// TIA Portal project "LIMIT" (V16)

(* hardware
DEVICE "S7-1200 station_1"  S7-1200 Station
   slot 0: "Rack_0"  S7-1200 Rack  Rack  V1.0
   slot 1: "PLC_1"  CPU 1212C AC/DC/Rly  6ES7 212-1BE40-0XB0  V4.4
*)

// ===== PLC "PLC_1"  CPU 1212C AC/DC/Rly =====

VAR_GLOBAL   // PLC tag table "Default tag table"
   "START" AT %I0.0 : Bool;
   "STOP" AT %I0.1 : Bool;
   "M1" AT %Q0.0 : Bool;
   "X" AT %M0.0 : Bool;
   "TM" AT %M0.1 : Bool;
   "L1" AT %I0.2 : Bool;
   "L2" AT %I0.3 : Bool;
   "L3" AT %I0.4 : Bool;
   "OFF" AT %M1.1 : Bool;
   "M2" AT %Q0.1 : Bool;
   "Tag_1" AT %M2.0 : Bool;
END_VAR

// folder: System blocks/Program resources

DATA_BLOCK "T"   // DB1
{ S7_Optimized_Access := 'TRUE' }
AUTHOR : Simatic
FAMILY : IEC
NAME : IEC_TMR
VERSION : 1.0
// stored: InstanceOfName IEC_TIMER
"IEC_TIMER"
BEGIN
END_DATA_BLOCK

// folder: (top level)

ORGANIZATION_BLOCK "Main"   // OB1, LAD, ProgramCycle
TITLE = "Main Program Sweep (Cycle)"
{ S7_Optimized_Access := 'TRUE' }
VERSION : 0.1
   VAR_INPUT
      Initial_Call : Bool;   // Initial call of this OB
      Remanence : Bool;   // =True, if remanent data are available
   END_VAR
   VAR_TEMP   // added for the SCL form of the ladder/FBD networks
      _w1 : Bool;
   END_VAR
BEGIN

REGION Network 1
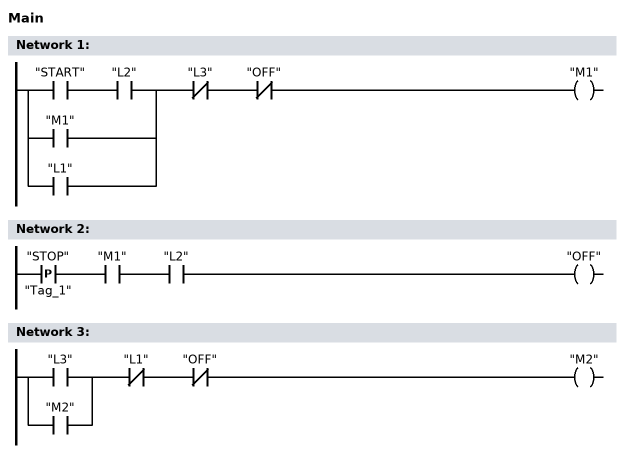
   RUNG wire#powerrail
      Contact( "START" )
      Contact( "L2" )
      wire#w1
      I_Contact( "L3" )
      I_Contact( "OFF" )
      Coil( "M1" )
   END_RUNG
   RUNG wire#powerrail
      Contact( "M1" )
   END_RUNG wire#w1
   RUNG wire#powerrail
      Contact( "L1" )
   END_RUNG wire#w1
   // the same network as SCL:
   "M1" := (("START" AND "L2") OR "M1" OR "L1") AND NOT "L3" AND NOT "OFF";
END_REGION

REGION Network 2
   RUNG wire#powerrail
      P_Contact(operand := "STOP", bit := "Tag_1")
      Contact( "M1" )
      Contact( "L2" )
      Coil( "OFF" )
   END_RUNG
   // the same network as SCL:
   #_w1 := "STOP" AND NOT "Tag_1";   // rising edge of "STOP"
   "Tag_1" := "STOP";
   "OFF" := #_w1 AND "M1" AND "L2";
END_REGION

REGION Network 3
   RUNG wire#powerrail
      Contact( "L3" )
      wire#w1
      I_Contact( "L1" )
      I_Contact( "OFF" )
      Coil( "M2" )
   END_RUNG
   RUNG wire#powerrail
      Contact( "M2" )
   END_RUNG wire#w1
   // the same network as SCL:
   "M2" := ("L3" OR "M2") AND NOT "L1" AND NOT "OFF";
END_REGION
END_ORGANIZATION_BLOCK